{attribute 'qualified_only'}
VAR_GLOBAL


END_VAR

(* stored: Version 1.1.0.1, ProductVersion 3.1.4024.12
   GVL GVL_IO: Id {0b120464-fa57-4150-9e08-41cfde9a87cd} *)
